SUBAPPLICATION Uebung_201b_AX (* Interlock: ILOCK_BLOCK_AX (Motor Rechts/Linkslauf via Adapter) *)
  (* Standard: 61499-2; Description: Copyright (c) 2023 Meisterschulen am Ostbahnhof This program and the accompanying materials are made available under the terms of the Eclipse Public License 2.0 which is available at https://www.eclipse.org/legal/epl-2.0/ SPDX-License-Identifier: EPL-2.0 *)
  (* Version 1.0, 2026-04-19, Franz Höpfinger, Meisterschulen am Ostbahnhof, initial API and implementation and/or initial documentation *)
  PACKAGE Uebungen;
  IMPORT logiBUS::io::DI::logiBUS_DI::Input_I1;
  IMPORT logiBUS::io::DI::logiBUS_DI::Input_I2;
  IMPORT logiBUS::io::DQ::logiBUS_DO::Output_Q5;
  IMPORT logiBUS::io::DQ::logiBUS_DO::Output_Q56;
  IMPORT logiBUS::io::DQ::logiBUS_DO::Output_Q6;
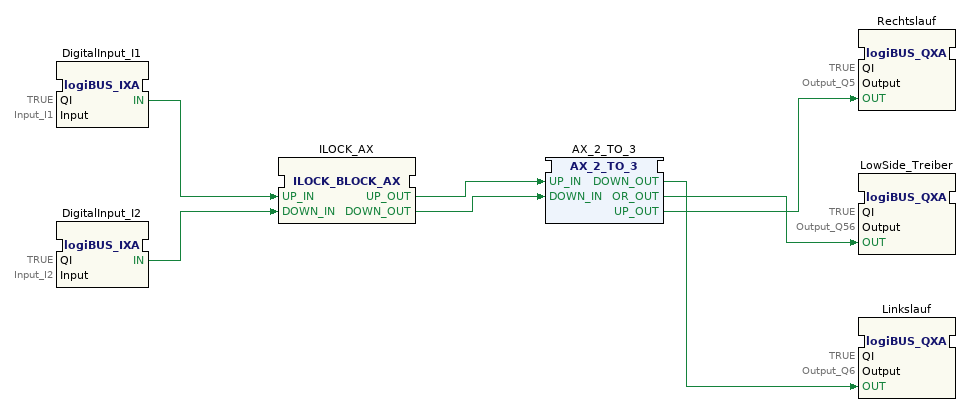
  FBS
    DigitalInput_I1 : logiBUS::io::DI::logiBUS_IXA(QI := TRUE, Input := Input_I1);
    DigitalInput_I2 : logiBUS::io::DI::logiBUS_IXA(QI := TRUE, Input := Input_I2);
    ILOCK_AX : logiBUS::signalprocessing::interlock::ILOCK_BLOCK_AX;
    Rechtslauf : logiBUS::io::DQ::logiBUS_QXA(QI := TRUE, Output := Output_Q5);
    LowSide_Treiber : logiBUS::io::DQ::logiBUS_QXA(QI := TRUE, Output := Output_Q56);
    Linkslauf : logiBUS::io::DQ::logiBUS_QXA(QI := TRUE, Output := Output_Q6);
  END_FBS
  SUBAPPS
    AX_2_TO_3 : MyLib::sys::AX_2_TO_3;
  END_SUBAPPS
  ADAPTER_CONNECTIONS
    DigitalInput_I1.IN TO ILOCK_AX.UP_IN;
    DigitalInput_I2.IN TO ILOCK_AX.DOWN_IN;
    AX_2_TO_3.DOWN_OUT TO Linkslauf.OUT;
    AX_2_TO_3.OR_OUT TO LowSide_Treiber.OUT;
    AX_2_TO_3.UP_OUT TO Rechtslauf.OUT;
    ILOCK_AX.UP_OUT TO AX_2_TO_3.UP_IN;
    ILOCK_AX.DOWN_OUT TO AX_2_TO_3.DOWN_IN;
  END_CONNECTIONS
END_SUBAPPLICATION
